(* PLC project STD_TEST, LOLITECH BREMIZ 1 *)
(* stored: contentDescription This tests as most as possible IEC standard library, companyURL www.lolitech.com, productRelease 1, creationDateTime 2007-07-07 11:58:26 *)

FUNCTION_BLOCK TEST_FROM_STRINGS
  VAR_INPUT
    IN1 : STRING;
    IN2 : STRING;
    TESTNR : INT;
  END_VAR
  VAR_OUTPUT
    INTRES : INT;
    NEXT_TEST : INT;
    TEST_NAME : STRING;
  END_VAR
  VAR  (* added by the conversion: wires and edge detectors of the diagram *)
    _LIMIT60_OUT : INT;
  END_VAR

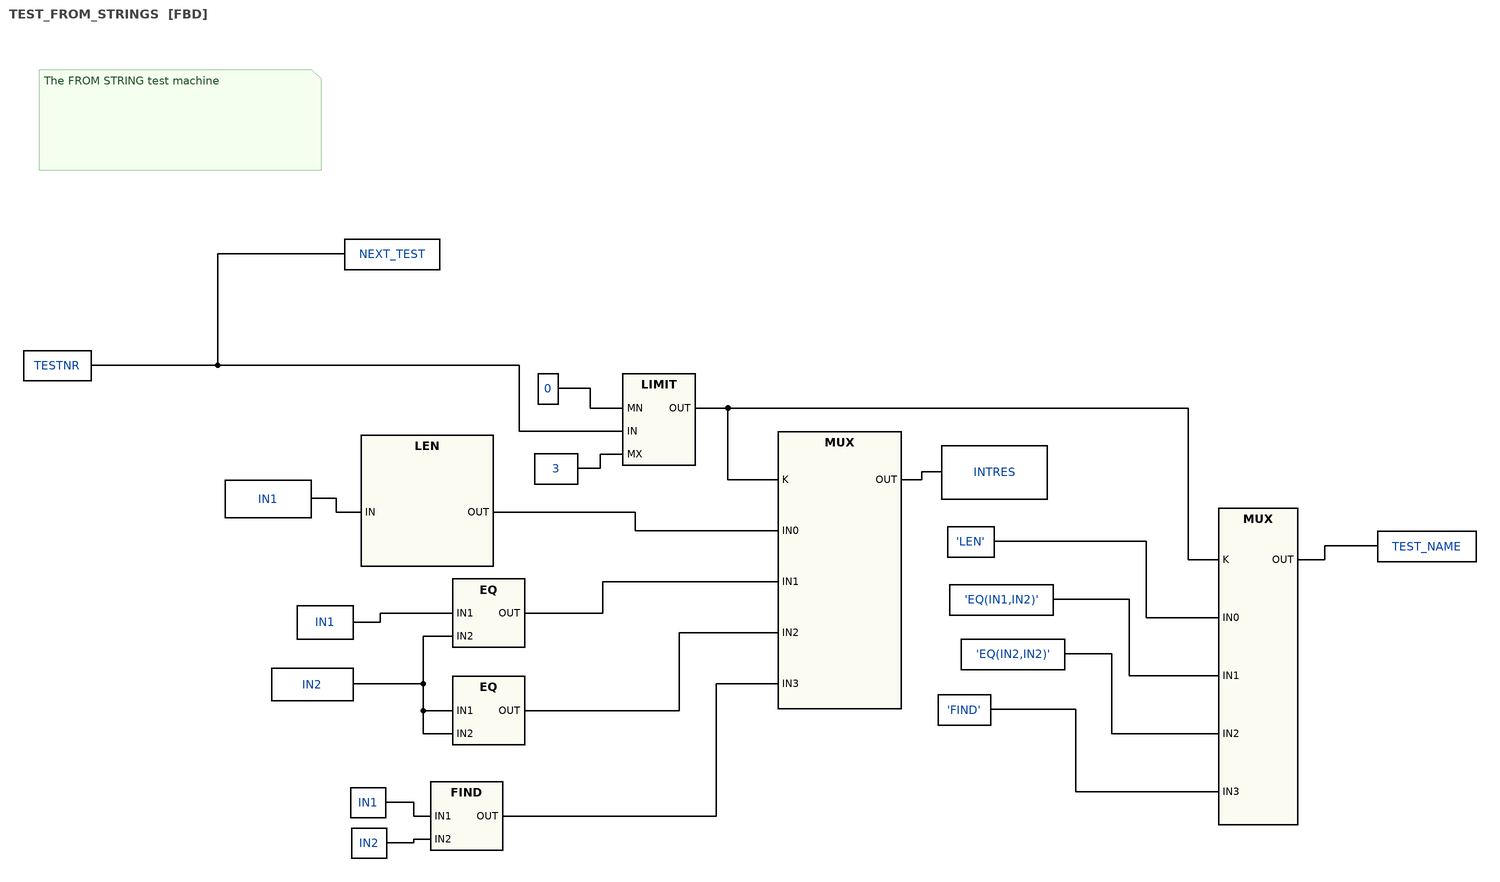
(* FBD diagram, written out as Structured Text *)
(* The FROM STRING test machine *)
NEXT_TEST := TESTNR;
_LIMIT60_OUT := LIMIT(0, TESTNR, 3);
INTRES := MUX(_LIMIT60_OUT, LEN(IN1), IN1 = IN2, IN2 = IN2, FIND(IN1, IN2));
TEST_NAME := MUX(_LIMIT60_OUT, 'LEN', 'EQ(IN1,IN2)', 'EQ(IN2,IN2)', 'FIND');
END_FUNCTION_BLOCK

FUNCTION_BLOCK TEST_STRINGS_OPS
  VAR_INPUT
    IN1 : STRING;
    IN2 : STRING;
    IN3 : STRING;
    TESTNR : INT;
    K : INT;
    P : INT;
    L : INT;
  END_VAR
  VAR_OUTPUT
    STRRES : STRING;
    NEXT_TEST : INT;
    TEST_NAME : STRING;
  END_VAR
  VAR  (* added by the conversion: wires and edge detectors of the diagram *)
    _LIMIT81_OUT : INT;
  END_VAR

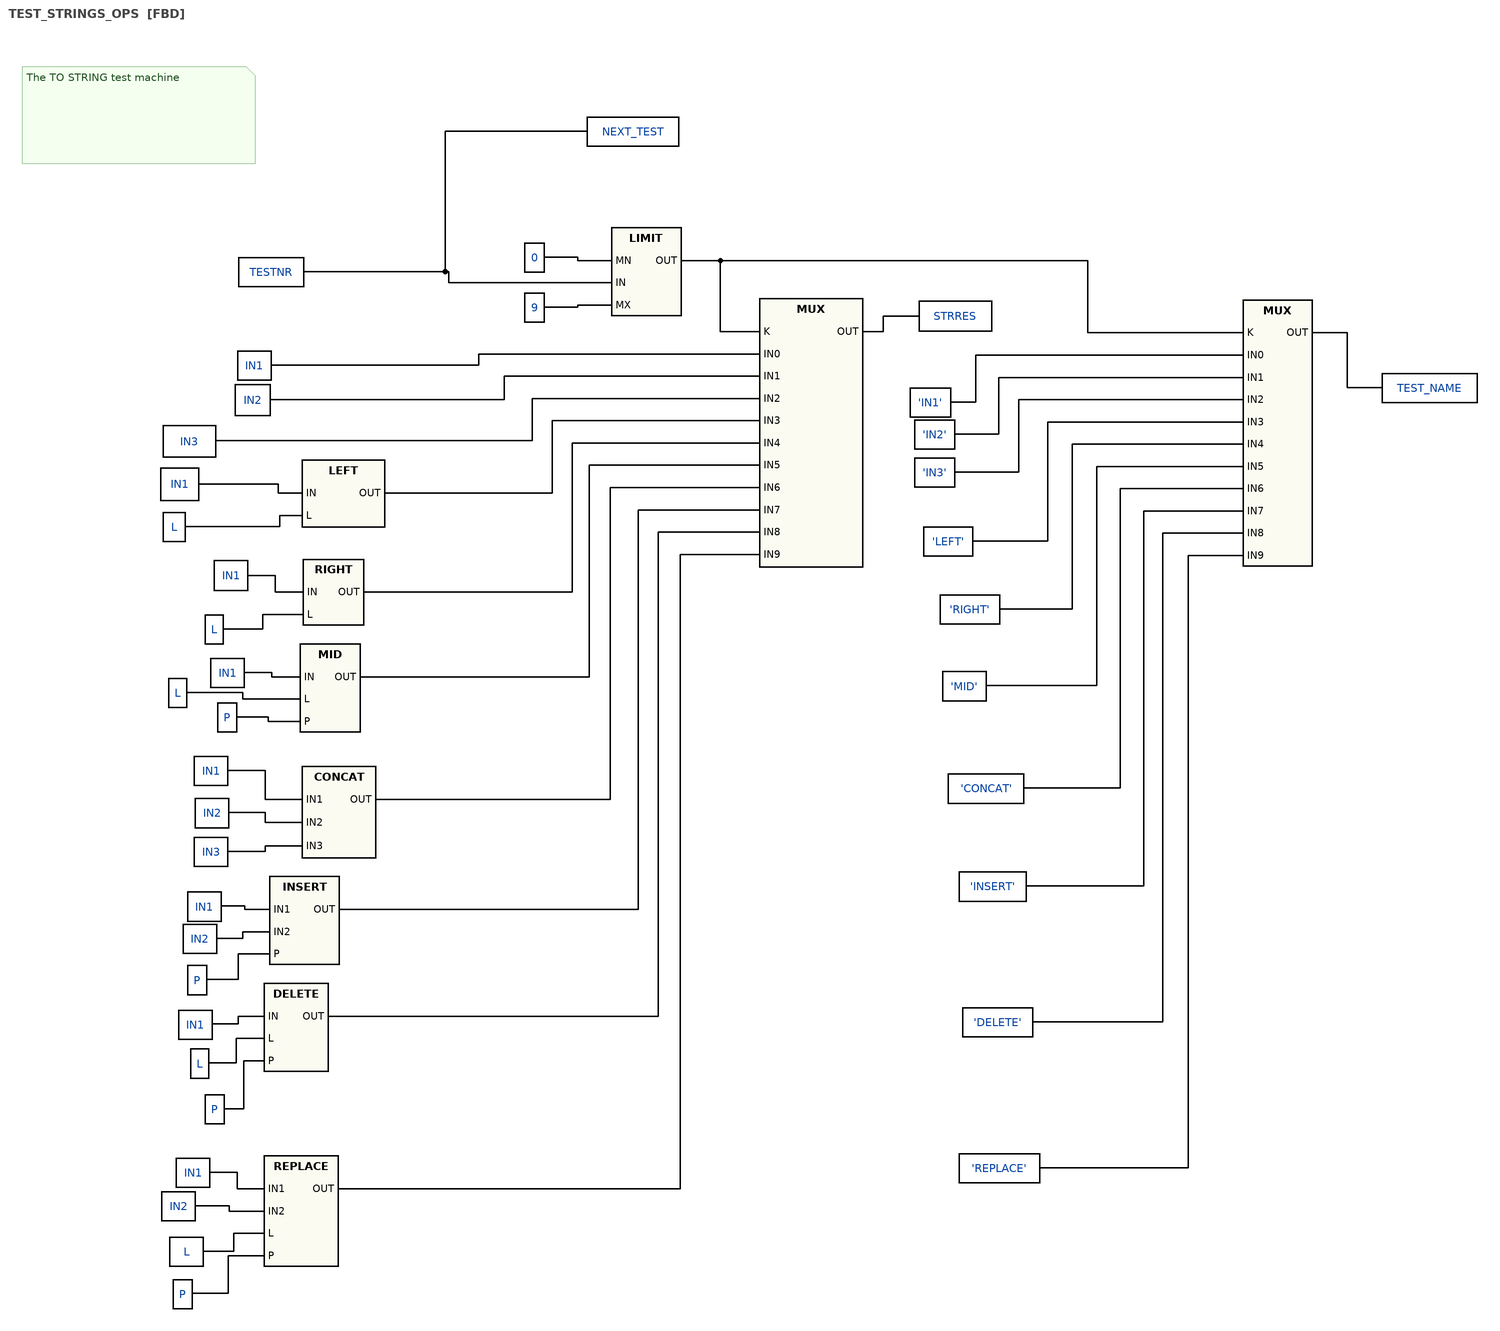
(* FBD diagram, written out as Structured Text *)
(* The TO STRING test machine *)
NEXT_TEST := TESTNR;
_LIMIT81_OUT := LIMIT(0, TESTNR, 9);
STRRES := MUX(_LIMIT81_OUT, IN1, IN2, IN3, LEFT(IN1, L), RIGHT(IN1, L), MID(IN1, L, P), CONCAT(IN1, IN2, IN3), INSERT(IN1, IN2, P), DELETE(IN1, L, P), REPLACE(IN1, IN2, L, P));
TEST_NAME := MUX(_LIMIT81_OUT, 'IN1', 'IN2', 'IN3', 'LEFT', 'RIGHT', 'MID', 'CONCAT', 'INSERT', 'DELETE', 'REPLACE');
END_FUNCTION_BLOCK

FUNCTION_BLOCK TEST_TO_STRINGS
  VAR_INPUT
    TESTNR : INT;
  END_VAR
  VAR_OUTPUT
    RES_STR : STRING;
    NEXT_TEST : INT;
    TEST_NAME : STRING;
    RES_BOOL : BOOL;
  END_VAR
  VAR  (* added by the conversion: wires and edge detectors of the diagram *)
    _LIMIT41_OUT : INT;
    _SINT_TO_STRING2_OUT : STRING;
    _INT_TO_STRING3_OUT : STRING;
    _DINT_TO_STRING4_OUT : STRING;
    _LINT_TO_STRING5_OUT : STRING;
    _USINT_TO_STRING6_OUT : STRING;
    _UINT_TO_STRING7_OUT : STRING;
    _UDINT_TO_STRING8_OUT : STRING;
    _ULINT_TO_STRING9_OUT : STRING;
    _REAL_TO_STRING10_OUT : STRING;
    _LREAL_TO_STRING11_OUT : STRING;
    _TIME_TO_STRING12_OUT : STRING;
    _DATE_TO_STRING13_OUT : STRING;
    _TOD_TO_STRING14_OUT : STRING;
    _DT_TO_STRING35_OUT : STRING;
    _BYTE_TO_STRING15_OUT : STRING;
    _WORD_TO_STRING16_OUT : STRING;
    _DWORD_TO_STRING17_OUT : STRING;
    _LWORD_TO_STRING18_OUT : STRING;
    _BOOL_TO_STRING1_OUT : STRING;
  END_VAR

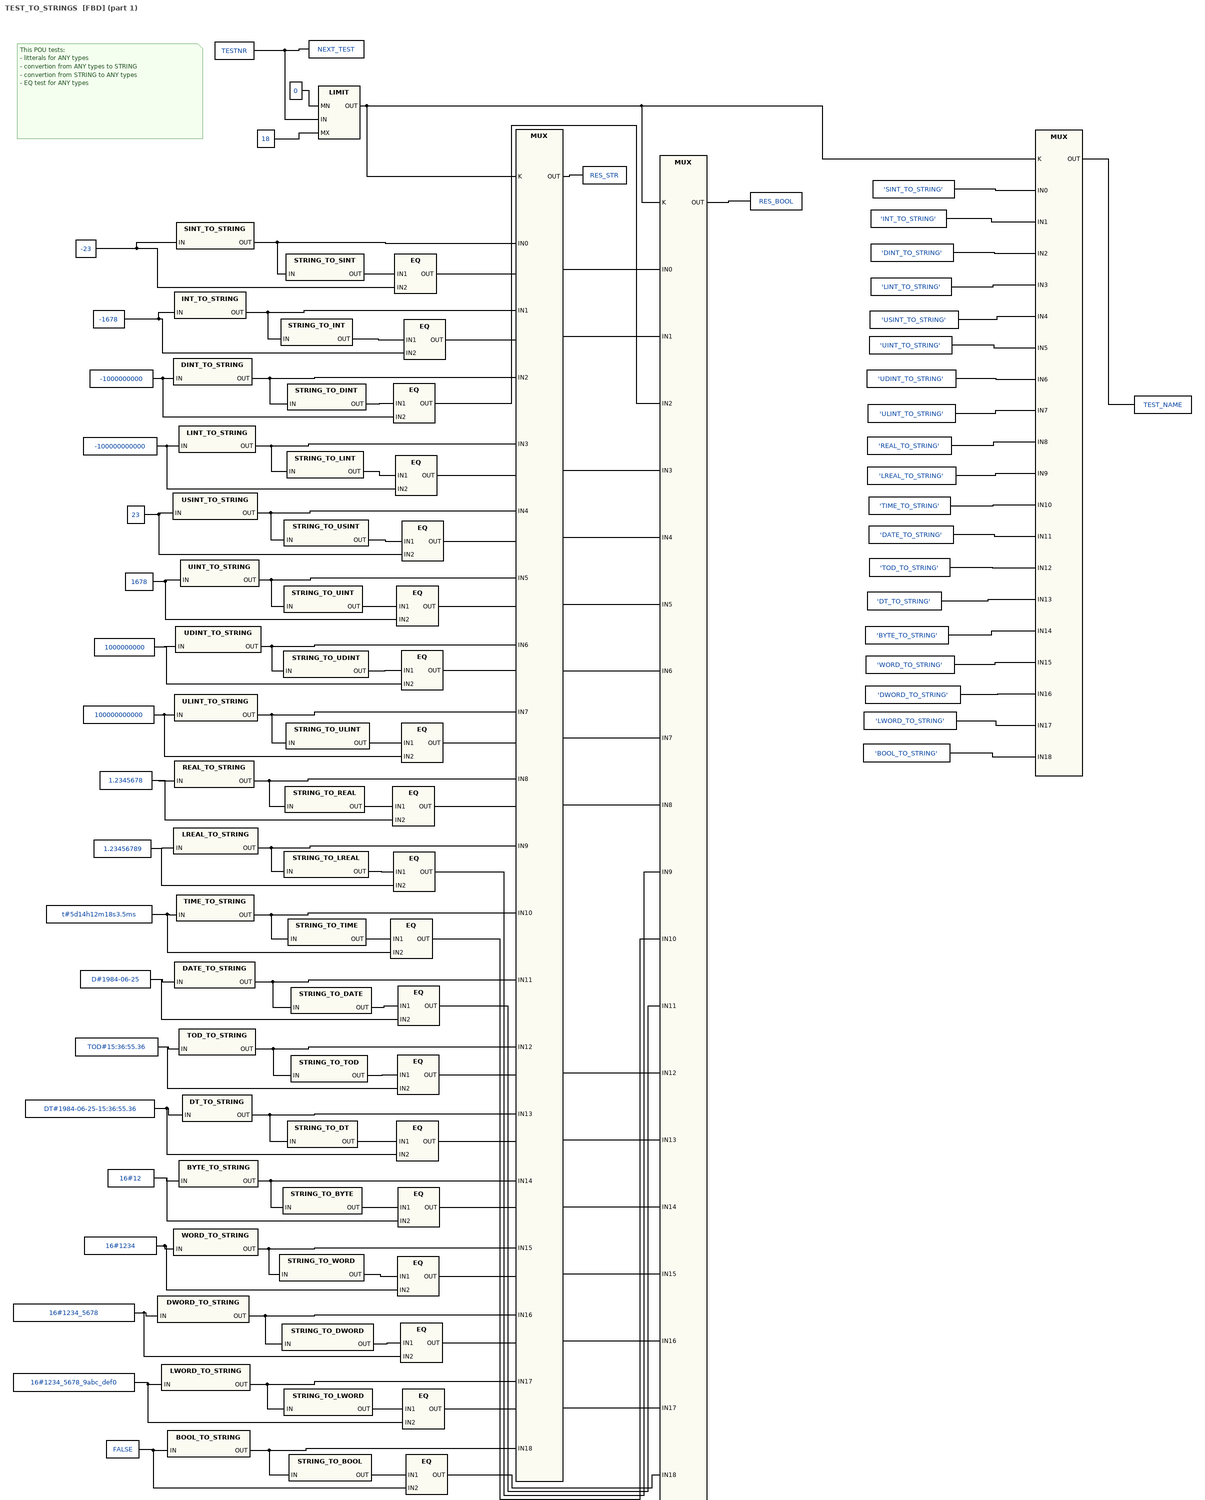
(* FBD diagram, written out as Structured Text *)
(* This POU tests:
- litterals for ANY types
- convertion from ANY types to STRING
- convertion from STRING to ANY types
- EQ test for ANY types *)
NEXT_TEST := TESTNR;
_LIMIT41_OUT := LIMIT(0, TESTNR, 18);
_SINT_TO_STRING2_OUT := SINT_TO_STRING(-23);
_INT_TO_STRING3_OUT := INT_TO_STRING(-1678);
_DINT_TO_STRING4_OUT := DINT_TO_STRING(-1000000000);
_LINT_TO_STRING5_OUT := LINT_TO_STRING(-100000000000);
_USINT_TO_STRING6_OUT := USINT_TO_STRING(23);
_UINT_TO_STRING7_OUT := UINT_TO_STRING(1678);
_UDINT_TO_STRING8_OUT := UDINT_TO_STRING(1000000000);
_ULINT_TO_STRING9_OUT := ULINT_TO_STRING(100000000000);
_REAL_TO_STRING10_OUT := REAL_TO_STRING(1.2345678);
_LREAL_TO_STRING11_OUT := LREAL_TO_STRING(1.23456789);
_TIME_TO_STRING12_OUT := TIME_TO_STRING(t#5d14h12m18s3.5ms);
_DATE_TO_STRING13_OUT := DATE_TO_STRING(D#1984-06-25);
_TOD_TO_STRING14_OUT := TOD_TO_STRING(TOD#15:36:55.36);
_DT_TO_STRING35_OUT := DT_TO_STRING(DT#1984-06-25-15:36:55.36);
_BYTE_TO_STRING15_OUT := BYTE_TO_STRING(16#12);
_WORD_TO_STRING16_OUT := WORD_TO_STRING(16#1234);
_DWORD_TO_STRING17_OUT := DWORD_TO_STRING(16#1234_5678);
_LWORD_TO_STRING18_OUT := LWORD_TO_STRING(16#1234_5678_9abc_def0);
_BOOL_TO_STRING1_OUT := BOOL_TO_STRING(FALSE);
RES_STR := MUX(_LIMIT41_OUT, _SINT_TO_STRING2_OUT, _INT_TO_STRING3_OUT, _DINT_TO_STRING4_OUT, _LINT_TO_STRING5_OUT, _USINT_TO_STRING6_OUT, _UINT_TO_STRING7_OUT, _UDINT_TO_STRING8_OUT, _ULINT_TO_STRING9_OUT, _REAL_TO_STRING10_OUT, _LREAL_TO_STRING11_OUT, _TIME_TO_STRING12_OUT, _DATE_TO_STRING13_OUT, _TOD_TO_STRING14_OUT, _DT_TO_STRING35_OUT, _BYTE_TO_STRING15_OUT, _WORD_TO_STRING16_OUT, _DWORD_TO_STRING17_OUT, _LWORD_TO_STRING18_OUT, _BOOL_TO_STRING1_OUT);
RES_BOOL := MUX(_LIMIT41_OUT, STRING_TO_SINT(_SINT_TO_STRING2_OUT) = (-23), STRING_TO_INT(_INT_TO_STRING3_OUT) = (-1678), STRING_TO_DINT(_DINT_TO_STRING4_OUT) = (-1000000000), STRING_TO_LINT(_LINT_TO_STRING5_OUT) = (-100000000000), STRING_TO_USINT(_USINT_TO_STRING6_OUT) = 23, STRING_TO_UINT(_UINT_TO_STRING7_OUT) = 1678, STRING_TO_UDINT(_UDINT_TO_STRING8_OUT) = 1000000000, STRING_TO_ULINT(_ULINT_TO_STRING9_OUT) = 100000000000, STRING_TO_REAL(_REAL_TO_STRING10_OUT) = 1.2345678, STRING_TO_LREAL(_LREAL_TO_STRING11_OUT) = 1.23456789, STRING_TO_TIME(_TIME_TO_STRING12_OUT) = t#5d14h12m18s3.5ms, STRING_TO_DATE(_DATE_TO_STRING13_OUT) = (D#1984-06-25), STRING_TO_TOD(_TOD_TO_STRING14_OUT) = TOD#15:36:55.36, STRING_TO_DT(_DT_TO_STRING35_OUT) = (DT#1984-06-25-15:36:55.36), STRING_TO_BYTE(_BYTE_TO_STRING15_OUT) = 16#12, STRING_TO_WORD(_WORD_TO_STRING16_OUT) = 16#1234, STRING_TO_DWORD(_DWORD_TO_STRING17_OUT) = 16#1234_5678, STRING_TO_LWORD(_LWORD_TO_STRING18_OUT) = 16#1234_5678_9abc_def0, STRING_TO_BOOL(_BOOL_TO_STRING1_OUT) = FALSE);
TEST_NAME := MUX(_LIMIT41_OUT, 'SINT_TO_STRING', 'INT_TO_STRING', 'DINT_TO_STRING', 'LINT_TO_STRING', 'USINT_TO_STRING', 'UINT_TO_STRING', 'UDINT_TO_STRING', 'ULINT_TO_STRING', 'REAL_TO_STRING', 'LREAL_TO_STRING', 'TIME_TO_STRING', 'DATE_TO_STRING', 'TOD_TO_STRING', 'DT_TO_STRING', 'BYTE_TO_STRING', 'WORD_TO_STRING', 'DWORD_TO_STRING', 'LWORD_TO_STRING', 'BOOL_TO_STRING');
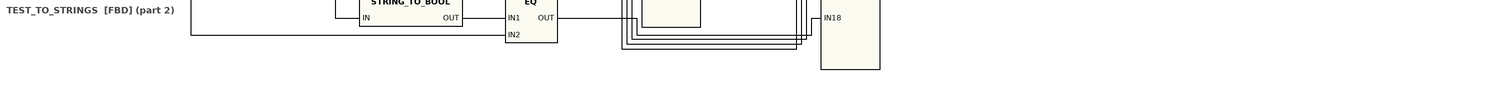
END_FUNCTION_BLOCK

PROGRAM MAIN_TEST
  VAR
    STR1 : STRING := '3.456789';
    INT1 : INT := 1;
  END_VAR
  VAR
    RES_TO_STR AT %QB0 : STRING;
    RES_FROM_STR AT %QW1 : INT;
    TEST_NB AT %IW0 : INT := 0;
  END_VAR
  VAR_EXTERNAL
    TO_STR_TEST_NAME : STRING;
    FROM_STR_TEST_NAME : STRING;
  END_VAR
  VAR
    RES_STR_OPS AT %QB3 : STRING;
    STR_OPS_TEST_NAME AT %QB4 : STRING;
    RES_TO_STR_BOOL AT %QX7 : BOOL;
  END_VAR

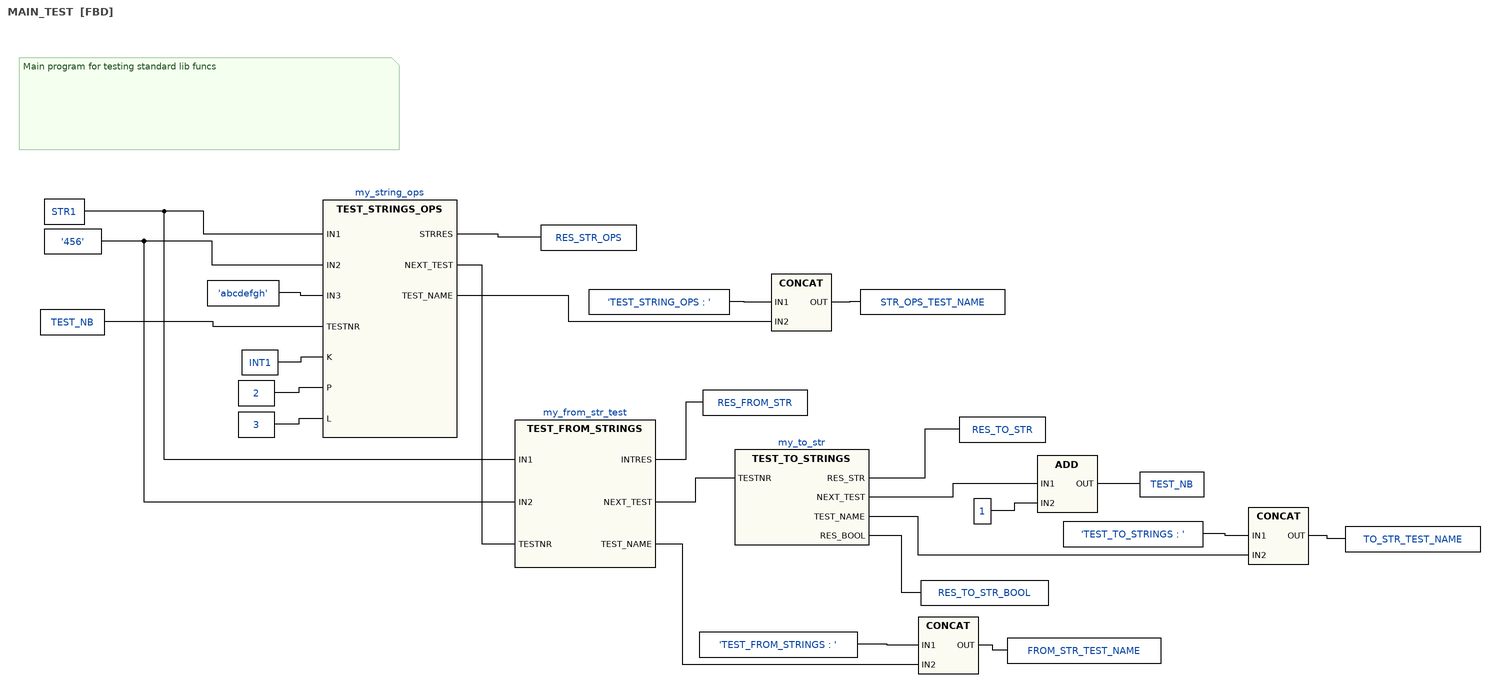
(* FBD diagram, written out as Structured Text *)
(* Main program for testing standard lib funcs *)
my_string_ops(IN1 := STR1, IN2 := '456', IN3 := 'abcdefgh', TESTNR := TEST_NB, K := INT1, P := 2, L := 3);
RES_STR_OPS := my_string_ops.STRRES;
STR_OPS_TEST_NAME := CONCAT('TEST_STRING_OPS : ', my_string_ops.TEST_NAME);
my_from_str_test(IN1 := STR1, IN2 := '456', TESTNR := my_string_ops.NEXT_TEST);
RES_FROM_STR := my_from_str_test.INTRES;
my_to_str(TESTNR := my_from_str_test.NEXT_TEST);
RES_TO_STR := my_to_str.RES_STR;
TEST_NB := my_to_str.NEXT_TEST + 1;
TO_STR_TEST_NAME := CONCAT('TEST_TO_STRINGS : ', my_to_str.TEST_NAME);
RES_TO_STR_BOOL := my_to_str.RES_BOOL;
FROM_STR_TEST_NAME := CONCAT('TEST_FROM_STRINGS : ', my_from_str_test.TEST_NAME);
END_PROGRAM

CONFIGURATION STD_CONF
  VAR_GLOBAL
    TO_STR_TEST_NAME AT %QB2 : STRING := 'str test name';
  END_VAR
  RESOURCE STD_RESSOURCE ON PLC
    VAR_GLOBAL
      FROM_STR_TEST_NAME AT %QB10 : STRING;
    END_VAR
    TASK STD_TASK(INTERVAL := 00:00:00.100000, PRIORITY := 0);
    PROGRAM MAIN_INSTANCE : MAIN_TEST;
  END_RESOURCE
END_CONFIGURATION
